(* CODESYS project Burner.project
   Title: Burner
   Version: 0.0.0.0
   Author: Plinfa7

Project tree, tasks and I/O mapping:
  MyController : TM241CEC24T/U, Schneider Electric, order no. TM241CEC24T/U, version 4.0.5.9
    application Application
      task MAST (cyclic, interval 20 ms, priority 15, watchdog 100 ms x 1) calls POU_modbus_READ_VAR, POU_modbus_WRITE_VAR_bit, POU_modbus_SINGLE_WRITE, POU_test
      global variables GVL
      program POU_test [LD]
      Symbols
    DI : Digital Inputs, Schneider Electric, version 4.0.5.9
        input  iwDI_IW0 : WORD  // IW0
        input  ibDI_IB1 : BYTE  // IB1
    DQ : Digital Outputs, Schneider Electric, version 4.0.5.9
        output qwDQ_QW0 : WORD  // QW0
        output qbDQ_QB1 : BYTE  // QB1
    Counters : Counters, Schneider Electric, version 4.0.5.9
    Pulse_Generators : Pulse Generators, Schneider Electric, version 4.0.5.9
    Cartridge_1 : Cartridge, Schneider Electric, version 4.0.5.9
    IO_Bus : IO bus - TM3, Schneider Electric, version 4.0.5.9
      A2 : TM3DI32K, Schneider Electric, order no. TM3DI32K, version 1.0.1.2
          unmapped channels: ID0
      A3 : TM3DI32K, Schneider Electric, order no. TM3DI32K, version 1.0.1.2
          input  idwModule_1_ID0 : DWORD  // ID0
      A6 : TM3DQ32TK, Schneider Electric, order no. TM3DQ32TK, version 1.0.1.2
          output qdwModule_2_QD0 : DWORD  // QD0
      A4 : TM3DQ32TK, Schneider Electric, order no. TM3DQ32TK, version 1.0.1.2
          output KL01 : BOOL  // QD0.Q0
          output KL02 : BOOL  // QD0.Q1
          output KL03 : BOOL  // QD0.Q2
          output KL04 : BOOL  // QD0.Q3
          output KL05 : BOOL  // QD0.Q4
          output KL06 : BOOL  // QD0.Q5
          output KL07 : BOOL  // QD0.Q6
          output KL08 : BOOL  // QD0.Q7
          output KL09 : BOOL  // QD0.Q8
          output KL10 : BOOL  // QD0.Q9
          output KL11 : BOOL  // QD0.Q10
          output KL12 : BOOL  // QD0.Q11
          output KL13 : BOOL  // QD0.Q12
          output KL14 : BOOL  // QD0.Q13
          output KL15 : BOOL  // QD0.Q14
          output KL16 : BOOL  // QD0.Q15
          output KL17 : BOOL  // QD0.Q16
          output KL18 : BOOL  // QD0.Q17
          output KL19 : BOOL  // QD0.Q18
          output KL20 : BOOL  // QD0.Q19
          output KL21 : BOOL  // QD0.Q20
          output KL22 : BOOL  // QD0.Q21
          output KL23 : BOOL  // QD0.Q22
          output KL24 : BOOL  // QD0.Q23
          output KL25 : BOOL  // QD0.Q24
          output KL26 : BOOL  // QD0.Q25
          output KL27 : BOOL  // QD0.Q26
          output KL28 : BOOL  // QD0.Q27
          output KL29 : BOOL  // QD0.Q28
          output KL30 : BOOL  // QD0.Q29
          output KL31 : BOOL  // QD0.Q30
          output KL32 : BOOL  // QD0.Q31
          unmapped channels: QD0
      A5 : TM3DQ32TK, Schneider Electric, order no. TM3DQ32TK, version 1.0.1.2
          output qdwA4_1_QD0_1 : DWORD  // QD0
    COM_Bus : COM bus, Schneider Electric, version 4.0.5.9
    Ethernet_1 : Ethernet Network, Schneider Electric, version 4.0.5.9
    Serial_Line_1 : Serial line, Schneider Electric, version 4.0.5.9 (disabled)
    Serial_Line_2 : Serial line, Schneider Electric, version 4.0.5.9
      Modbus_Manager : Modbus Manager, Schneider Electric, version 4.0.0.2
    CAN_1 : CANopen bus, Schneider Electric, version 4.0.5.9 (disabled)
  HMIGTO5310_5315 : HMIGTO5310/5315, Schneider Electric, order no. HMIGTO5310/5315, version 3.5.3.55
    HMI Application
    COM1
      SoMachine_Network_Manager : SoMachine-Network Manager, Schneider Electric, version 4.0.0.2
    COM2
      SoMachine_Network_Manager1 : SoMachine-Network Manager, Schneider Electric, version 4.0.0.2
    Ethernet
      SoMachine_Network_Manager2 : SoMachine-Network Manager, Schneider Electric, version 4.0.0.2
    USB
      SoMachine_Network_Manager3 : SoMachine-Network Manager, Schneider Electric, version 4.0.0.2
  program POU_modbus_SINGLE_WRITE [LD]
  program POU_modbus_READ_VAR [LD]
  program POU_modbus_WRITE_VAR_bit [FBD]
  Vijeo Designer Project Container Data
  Vijeo Designer Project Container
*)

// MyController/Application/GVL
VAR_GLOBAL
	KLxx_ON_OFF: BOOL;
END_VAR

// POU_modbus_READ_VAR
PROGRAM POU_modbus_READ_VAR
VAR
	temp_var: BOOL;
	res_var: BOOL;
	ADDM_REG0: ADDM;
	SLI_Slave_addr: ADDRESS;
	start: BOOL;
	READ_VAR_REG0: READ_VAR;
	ReceiveBuffer: ARRAY [0..4] OF WORD;
	BLINK_0: BLINK;
	go: BOOL;
END_VAR

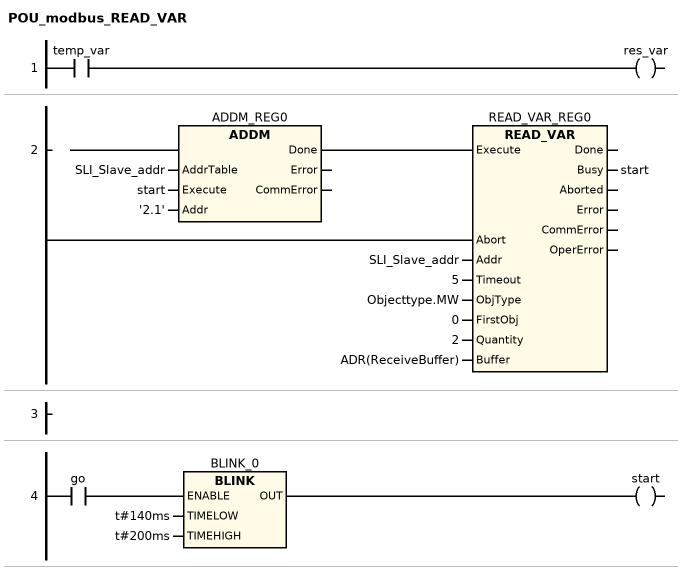
// NETWORK 1
res_var := temp_var;

// NETWORK 2
//   Objecttype.MW: Internal Register
ADDM_REG0(AddrTable := SLI_Slave_addr, Execute := start, Addr := '2.1'); // ADDM
READ_VAR_REG0(
    Execute := ADDM_REG0.Done,
    Abort := TRUE,
    Addr := SLI_Slave_addr,
    Timeout := 5,
    ObjType := Objecttype.MW,
    FirstObj := 0,
    Quantity := 2,
    Buffer := ADR(ReceiveBuffer),
    Busy => start); // READ_VAR

// NETWORK 3

// NETWORK 4
BLINK_0(ENABLE := go, TIMELOW := t#140ms, TIMEHIGH := t#200ms); // BLINK
start := BLINK_0.OUT;

END_PROGRAM

// POU_modbus_WRITE_VAR_bit
PROGRAM POU_modbus_WRITE_VAR_bit
VAR
	ADDM_REG0: ADDM;
	SLI_Slave_addr: ADDRESS;
	start: BOOL;
	SendBuffer: WORD := 1;
	SendBuffer2: ARRAY [0..3] OF WORD;
	BLINK_0: BLINK;
	WRITE_VAR_BIT: WRITE_VAR;
	go: BOOL := TRUE;
END_VAR
VAR // added by the converter: edge detectors and wires of the graphical bodies
    _rt1 : R_TRIG;
    _w1 : BOOL;
END_VAR

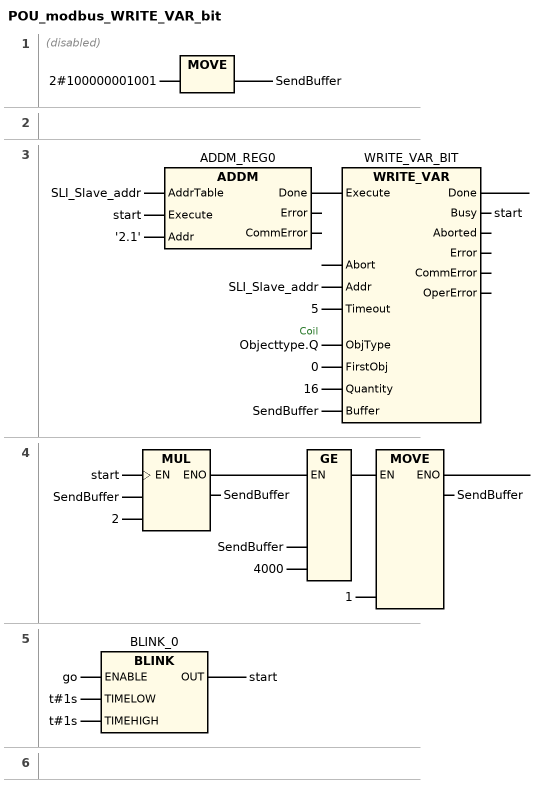
// NETWORK 1 (disabled)
// SendBuffer := 2#100000001001;

// NETWORK 2

// NETWORK 3
//   Objecttype.Q: Coil
ADDM_REG0(AddrTable := SLI_Slave_addr, Execute := start, Addr := '2.1'); // ADDM
WRITE_VAR_BIT(
    Execute := ADDM_REG0.Done,
    Addr := SLI_Slave_addr,
    Timeout := 5,
    ObjType := Objecttype.Q,
    FirstObj := 0,
    Quantity := 16,
    Buffer := SendBuffer,
    Busy => start); // WRITE_VAR

// NETWORK 4
_rt1(CLK := start);
_w1 := _rt1.Q;
IF _w1 THEN SendBuffer := SendBuffer * 2; END_IF
IF _w1 AND SendBuffer >= 4000 THEN SendBuffer := 1; END_IF

// NETWORK 5
BLINK_0(ENABLE := go, TIMELOW := t#1s, TIMEHIGH := t#1s); // BLINK
start := BLINK_0.OUT;

// NETWORK 6

END_PROGRAM

// POU_modbus_SINGLE_WRITE
PROGRAM POU_modbus_SINGLE_WRITE
VAR
	temp_var: BOOL;
	res_var: BOOL;
	ADDM_REG0: ADDM;
	SLI_Slave_addr: ADDRESS;
	start: BOOL;
	READ_VAR_REG0: READ_VAR;
	ReceiveBuffer: ARRAY [0..6] OF WORD;
	
	MV1_from_slave8 : WORD;
	MV2_from_slave8 : WORD;
	BLINK_0: BLINK;
	SINGLE_WRITE_REG0: SINGLE_WRITE;
	inc_val: WORD := 705;
	go: BOOL;
END_VAR
VAR // added by the converter: edge detectors and wires of the graphical bodies
    _rt1 : R_TRIG;
    _w1 : BOOL;
END_VAR

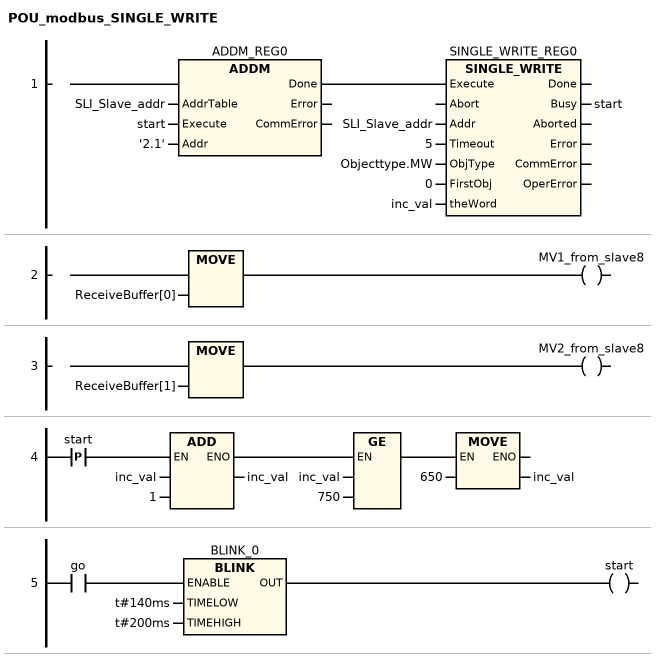
// NETWORK 1
//   Objecttype.MW: Internal Register
ADDM_REG0(AddrTable := SLI_Slave_addr, Execute := start, Addr := '2.1'); // ADDM
SINGLE_WRITE_REG0(
    Execute := ADDM_REG0.Done,
    Addr := SLI_Slave_addr,
    Timeout := 5,
    ObjType := Objecttype.MW,
    FirstObj := 0,
    theWord := inc_val,
    Busy => start); // SINGLE_WRITE

// NETWORK 2
MV1_from_slave8 := ReceiveBuffer[0];

// NETWORK 3
MV2_from_slave8 := ReceiveBuffer[1];

// NETWORK 4
_rt1(CLK := start);
_w1 := _rt1.Q;
IF _w1 THEN inc_val := inc_val + 1; END_IF
IF _w1 AND inc_val >= 750 THEN inc_val := 650; END_IF

// NETWORK 5
BLINK_0(ENABLE := go, TIMELOW := t#140ms, TIMEHIGH := t#200ms); // BLINK
start := BLINK_0.OUT;

END_PROGRAM

// MyController/Application/POU_test
PROGRAM POU_test
VAR
	led: BOOL;
END_VAR

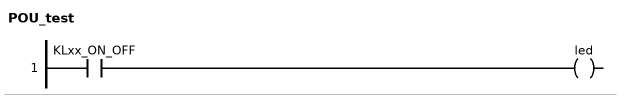
// NETWORK 1
led := KLxx_ON_OFF;

END_PROGRAM
